// TIA Portal V20 export
TYPE "UDT_Interlock_manual_STV"
   STRUCT
      "byte0.bit0" : Bool;
      "byte0.bit1" : Bool;
      Load_ok : Bool;
      "byte0.bit3" : Bool;
      "byte0.bit4" : Bool;
      "Byte0.bit8" : Bool;
      "Byte0.bit9" : Bool;
      Byte1_bit0 : Bool;
      Byte1_bit1 : Bool;
      Unload_ok : Bool;
      UnloadComplete : Bool;
      Byte1_bit8 : Bool;
      Byte1_bit9 : Bool;
      Byte1_bit10 : Bool;
      Byte1_bit6 : Bool;
      Byte1_bit7 : Bool;
   END_STRUCT;
END_TYPE
